(* CoDeSys 2.3 export: 6SHU-PV1.EXP *)

(* POU MAIN, CFC *)
PROGRAM MAIN
VAR
	TCT: ISTOK_TaskCycleTime;
END_VAR
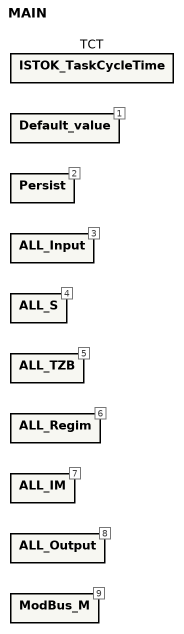
_CFC_ (* Continuous Function Chart, elements in execution order *)
#0 TCT:ISTOK_TaskCycleTime()
#1 Default_value()
#2 Persist()
#3 ALL_Input()
#4 ALL_S()
#5 ALL_TZB()
#6 ALL_Regim()
#7 ALL_IM()
#8 ALL_Output()
#9 ModBus_M()
_END_CFC_
(* the same logic as Structured Text *)
TCT();
Default_value();
Persist();
ALL_Input();
ALL_S();
ALL_TZB();
ALL_Regim();
ALL_IM();
ALL_Output();
ModBus_M();
END_PROGRAM

(* POU Lib/ISTOK_TaskCycleTime, CFC *)
FUNCTION_BLOCK ISTOK_TaskCycleTime
VAR_INPUT
END_VAR
VAR_OUTPUT
END_VAR
VAR
END_VAR
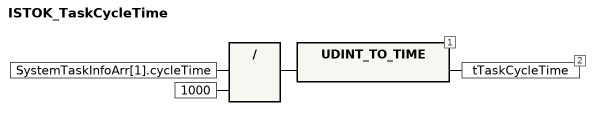
_CFC_ (* Continuous Function Chart, elements in execution order *)
#0 /(SystemTaskInfoArr[1].cycleTime, 1000)
#1 UDINT_TO_TIME(#0)
#2 tTaskCycleTime <= #1
_END_CFC_
END_FUNCTION_BLOCK

(* POU Default_value, CFC *)
PROGRAM Default_value
VAR
END_VAR
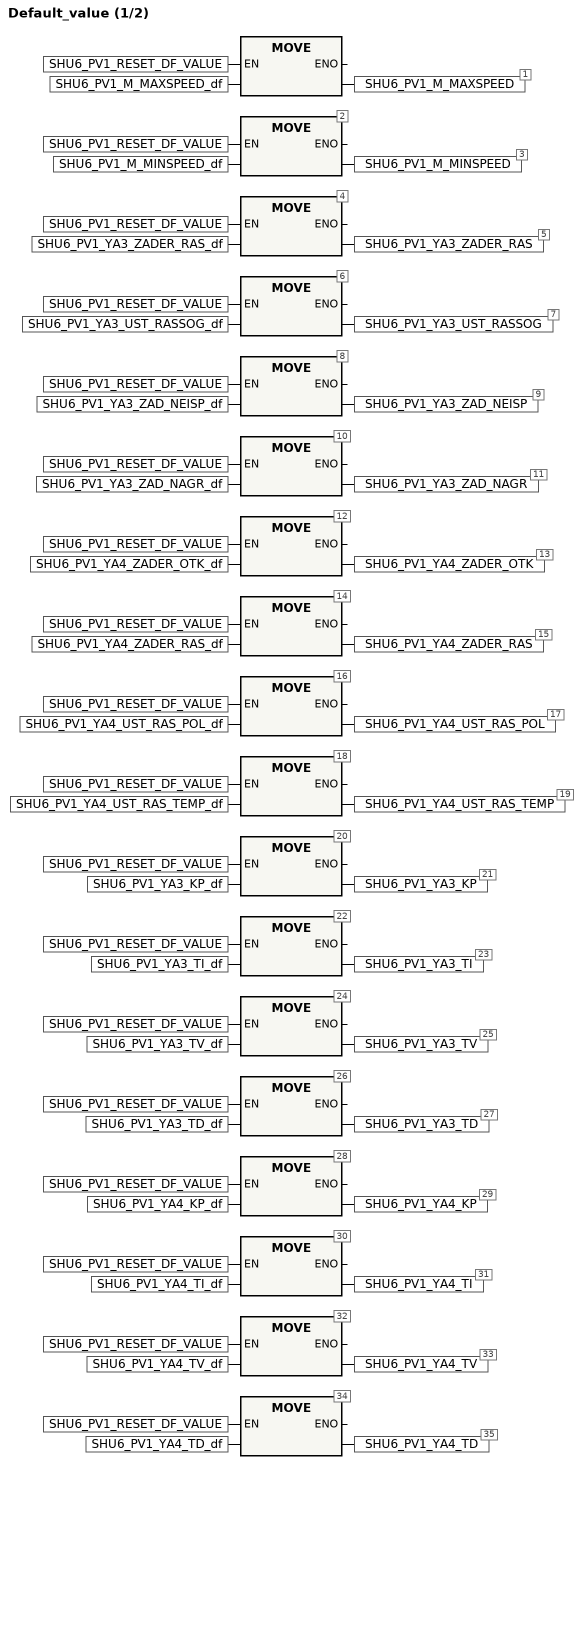
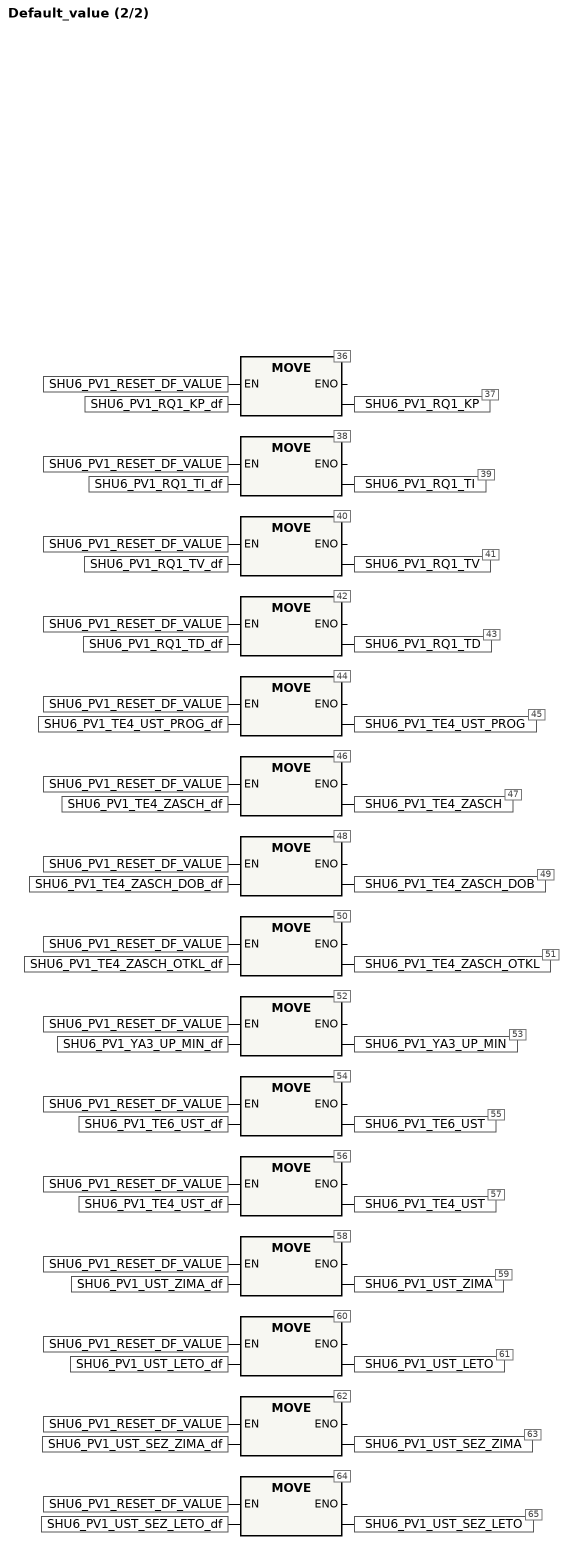
_CFC_ (* Continuous Function Chart, elements in execution order *)
#0 MOVE(EN: SHU6_PV1_RESET_DF_VALUE, SHU6_PV1_M_MAXSPEED_df)
#1 SHU6_PV1_M_MAXSPEED <= #0
#2 MOVE(EN: SHU6_PV1_RESET_DF_VALUE, SHU6_PV1_M_MINSPEED_df)
#3 SHU6_PV1_M_MINSPEED <= #2
#4 MOVE(EN: SHU6_PV1_RESET_DF_VALUE, SHU6_PV1_YA3_ZADER_RAS_df)
#5 SHU6_PV1_YA3_ZADER_RAS <= #4
#6 MOVE(EN: SHU6_PV1_RESET_DF_VALUE, SHU6_PV1_YA3_UST_RASSOG_df)
#7 SHU6_PV1_YA3_UST_RASSOG <= #6
#8 MOVE(EN: SHU6_PV1_RESET_DF_VALUE, SHU6_PV1_YA3_ZAD_NEISP_df)
#9 SHU6_PV1_YA3_ZAD_NEISP <= #8
#10 MOVE(EN: SHU6_PV1_RESET_DF_VALUE, SHU6_PV1_YA3_ZAD_NAGR_df)
#11 SHU6_PV1_YA3_ZAD_NAGR <= #10
#12 MOVE(EN: SHU6_PV1_RESET_DF_VALUE, SHU6_PV1_YA4_ZADER_OTK_df)
#13 SHU6_PV1_YA4_ZADER_OTK <= #12
#14 MOVE(EN: SHU6_PV1_RESET_DF_VALUE, SHU6_PV1_YA4_ZADER_RAS_df)
#15 SHU6_PV1_YA4_ZADER_RAS <= #14
#16 MOVE(EN: SHU6_PV1_RESET_DF_VALUE, SHU6_PV1_YA4_UST_RAS_POL_df)
#17 SHU6_PV1_YA4_UST_RAS_POL <= #16
#18 MOVE(EN: SHU6_PV1_RESET_DF_VALUE, SHU6_PV1_YA4_UST_RAS_TEMP_df)
#19 SHU6_PV1_YA4_UST_RAS_TEMP <= #18
#20 MOVE(EN: SHU6_PV1_RESET_DF_VALUE, SHU6_PV1_YA3_KP_df)
#21 SHU6_PV1_YA3_KP <= #20
#22 MOVE(EN: SHU6_PV1_RESET_DF_VALUE, SHU6_PV1_YA3_TI_df)
#23 SHU6_PV1_YA3_TI <= #22
#24 MOVE(EN: SHU6_PV1_RESET_DF_VALUE, SHU6_PV1_YA3_TV_df)
#25 SHU6_PV1_YA3_TV <= #24
#26 MOVE(EN: SHU6_PV1_RESET_DF_VALUE, SHU6_PV1_YA3_TD_df)
#27 SHU6_PV1_YA3_TD <= #26
#28 MOVE(EN: SHU6_PV1_RESET_DF_VALUE, SHU6_PV1_YA4_KP_df)
#29 SHU6_PV1_YA4_KP <= #28
#30 MOVE(EN: SHU6_PV1_RESET_DF_VALUE, SHU6_PV1_YA4_TI_df)
#31 SHU6_PV1_YA4_TI <= #30
#32 MOVE(EN: SHU6_PV1_RESET_DF_VALUE, SHU6_PV1_YA4_TV_df)
#33 SHU6_PV1_YA4_TV <= #32
#34 MOVE(EN: SHU6_PV1_RESET_DF_VALUE, SHU6_PV1_YA4_TD_df)
#35 SHU6_PV1_YA4_TD <= #34
#36 MOVE(EN: SHU6_PV1_RESET_DF_VALUE, SHU6_PV1_RQ1_KP_df)
#37 SHU6_PV1_RQ1_KP <= #36
#38 MOVE(EN: SHU6_PV1_RESET_DF_VALUE, SHU6_PV1_RQ1_TI_df)
#39 SHU6_PV1_RQ1_TI <= #38
#40 MOVE(EN: SHU6_PV1_RESET_DF_VALUE, SHU6_PV1_RQ1_TV_df)
#41 SHU6_PV1_RQ1_TV <= #40
#42 MOVE(EN: SHU6_PV1_RESET_DF_VALUE, SHU6_PV1_RQ1_TD_df)
#43 SHU6_PV1_RQ1_TD <= #42
#44 MOVE(EN: SHU6_PV1_RESET_DF_VALUE, SHU6_PV1_TE4_UST_PROG_df)
#45 SHU6_PV1_TE4_UST_PROG <= #44
#46 MOVE(EN: SHU6_PV1_RESET_DF_VALUE, SHU6_PV1_TE4_ZASCH_df)
#47 SHU6_PV1_TE4_ZASCH <= #46
#48 MOVE(EN: SHU6_PV1_RESET_DF_VALUE, SHU6_PV1_TE4_ZASCH_DOB_df)
#49 SHU6_PV1_TE4_ZASCH_DOB <= #48
#50 MOVE(EN: SHU6_PV1_RESET_DF_VALUE, SHU6_PV1_TE4_ZASCH_OTKL_df)
#51 SHU6_PV1_TE4_ZASCH_OTKL <= #50
#52 MOVE(EN: SHU6_PV1_RESET_DF_VALUE, SHU6_PV1_YA3_UP_MIN_df)
#53 SHU6_PV1_YA3_UP_MIN <= #52
#54 MOVE(EN: SHU6_PV1_RESET_DF_VALUE, SHU6_PV1_TE6_UST_df)
#55 SHU6_PV1_TE6_UST <= #54
#56 MOVE(EN: SHU6_PV1_RESET_DF_VALUE, SHU6_PV1_TE4_UST_df)
#57 SHU6_PV1_TE4_UST <= #56
#58 MOVE(EN: SHU6_PV1_RESET_DF_VALUE, SHU6_PV1_UST_ZIMA_df)
#59 SHU6_PV1_UST_ZIMA <= #58
#60 MOVE(EN: SHU6_PV1_RESET_DF_VALUE, SHU6_PV1_UST_LETO_df)
#61 SHU6_PV1_UST_LETO <= #60
#62 MOVE(EN: SHU6_PV1_RESET_DF_VALUE, SHU6_PV1_UST_SEZ_ZIMA_df)
#63 SHU6_PV1_UST_SEZ_ZIMA <= #62
#64 MOVE(EN: SHU6_PV1_RESET_DF_VALUE, SHU6_PV1_UST_SEZ_LETO_df)
#65 SHU6_PV1_UST_SEZ_LETO <= #64
_END_CFC_
(* the same logic as Structured Text *)
IF SHU6_PV1_RESET_DF_VALUE THEN SHU6_PV1_M_MAXSPEED := SHU6_PV1_M_MAXSPEED_df; END_IF;
IF SHU6_PV1_RESET_DF_VALUE THEN SHU6_PV1_M_MINSPEED := SHU6_PV1_M_MINSPEED_df; END_IF;
IF SHU6_PV1_RESET_DF_VALUE THEN SHU6_PV1_YA3_ZADER_RAS := SHU6_PV1_YA3_ZADER_RAS_df; END_IF;
IF SHU6_PV1_RESET_DF_VALUE THEN SHU6_PV1_YA3_UST_RASSOG := SHU6_PV1_YA3_UST_RASSOG_df; END_IF;
IF SHU6_PV1_RESET_DF_VALUE THEN SHU6_PV1_YA3_ZAD_NEISP := SHU6_PV1_YA3_ZAD_NEISP_df; END_IF;
IF SHU6_PV1_RESET_DF_VALUE THEN SHU6_PV1_YA3_ZAD_NAGR := SHU6_PV1_YA3_ZAD_NAGR_df; END_IF;
IF SHU6_PV1_RESET_DF_VALUE THEN SHU6_PV1_YA4_ZADER_OTK := SHU6_PV1_YA4_ZADER_OTK_df; END_IF;
IF SHU6_PV1_RESET_DF_VALUE THEN SHU6_PV1_YA4_ZADER_RAS := SHU6_PV1_YA4_ZADER_RAS_df; END_IF;
IF SHU6_PV1_RESET_DF_VALUE THEN SHU6_PV1_YA4_UST_RAS_POL := SHU6_PV1_YA4_UST_RAS_POL_df; END_IF;
IF SHU6_PV1_RESET_DF_VALUE THEN SHU6_PV1_YA4_UST_RAS_TEMP := SHU6_PV1_YA4_UST_RAS_TEMP_df; END_IF;
IF SHU6_PV1_RESET_DF_VALUE THEN SHU6_PV1_YA3_KP := SHU6_PV1_YA3_KP_df; END_IF;
IF SHU6_PV1_RESET_DF_VALUE THEN SHU6_PV1_YA3_TI := SHU6_PV1_YA3_TI_df; END_IF;
IF SHU6_PV1_RESET_DF_VALUE THEN SHU6_PV1_YA3_TV := SHU6_PV1_YA3_TV_df; END_IF;
IF SHU6_PV1_RESET_DF_VALUE THEN SHU6_PV1_YA3_TD := SHU6_PV1_YA3_TD_df; END_IF;
IF SHU6_PV1_RESET_DF_VALUE THEN SHU6_PV1_YA4_KP := SHU6_PV1_YA4_KP_df; END_IF;
IF SHU6_PV1_RESET_DF_VALUE THEN SHU6_PV1_YA4_TI := SHU6_PV1_YA4_TI_df; END_IF;
IF SHU6_PV1_RESET_DF_VALUE THEN SHU6_PV1_YA4_TV := SHU6_PV1_YA4_TV_df; END_IF;
IF SHU6_PV1_RESET_DF_VALUE THEN SHU6_PV1_YA4_TD := SHU6_PV1_YA4_TD_df; END_IF;
IF SHU6_PV1_RESET_DF_VALUE THEN SHU6_PV1_RQ1_KP := SHU6_PV1_RQ1_KP_df; END_IF;
IF SHU6_PV1_RESET_DF_VALUE THEN SHU6_PV1_RQ1_TI := SHU6_PV1_RQ1_TI_df; END_IF;
IF SHU6_PV1_RESET_DF_VALUE THEN SHU6_PV1_RQ1_TV := SHU6_PV1_RQ1_TV_df; END_IF;
IF SHU6_PV1_RESET_DF_VALUE THEN SHU6_PV1_RQ1_TD := SHU6_PV1_RQ1_TD_df; END_IF;
IF SHU6_PV1_RESET_DF_VALUE THEN SHU6_PV1_TE4_UST_PROG := SHU6_PV1_TE4_UST_PROG_df; END_IF;
IF SHU6_PV1_RESET_DF_VALUE THEN SHU6_PV1_TE4_ZASCH := SHU6_PV1_TE4_ZASCH_df; END_IF;
IF SHU6_PV1_RESET_DF_VALUE THEN SHU6_PV1_TE4_ZASCH_DOB := SHU6_PV1_TE4_ZASCH_DOB_df; END_IF;
IF SHU6_PV1_RESET_DF_VALUE THEN SHU6_PV1_TE4_ZASCH_OTKL := SHU6_PV1_TE4_ZASCH_OTKL_df; END_IF;
IF SHU6_PV1_RESET_DF_VALUE THEN SHU6_PV1_YA3_UP_MIN := SHU6_PV1_YA3_UP_MIN_df; END_IF;
IF SHU6_PV1_RESET_DF_VALUE THEN SHU6_PV1_TE6_UST := SHU6_PV1_TE6_UST_df; END_IF;
IF SHU6_PV1_RESET_DF_VALUE THEN SHU6_PV1_TE4_UST := SHU6_PV1_TE4_UST_df; END_IF;
IF SHU6_PV1_RESET_DF_VALUE THEN SHU6_PV1_UST_ZIMA := SHU6_PV1_UST_ZIMA_df; END_IF;
IF SHU6_PV1_RESET_DF_VALUE THEN SHU6_PV1_UST_LETO := SHU6_PV1_UST_LETO_df; END_IF;
IF SHU6_PV1_RESET_DF_VALUE THEN SHU6_PV1_UST_SEZ_ZIMA := SHU6_PV1_UST_SEZ_ZIMA_df; END_IF;
IF SHU6_PV1_RESET_DF_VALUE THEN SHU6_PV1_UST_SEZ_LETO := SHU6_PV1_UST_SEZ_LETO_df; END_IF;
END_PROGRAM

(* POU Persist, ST *)
PROGRAM Persist
VAR
	Save: WritePersistentData;
END_VAR
Save(NETID:='10.150.0.24.1.1',PORT:=801,START:=TRUE,TMOUT:=t#1s ,BUSY=> ,ERR=> ,	ERRID=> );
Save(NETID:='10.150.0.24.1.1',PORT:=801,START:= FALSE ,TMOUT:=t#1s ,BUSY=> ,ERR=> ,ERRID=> );
END_PROGRAM

(* POU Input/ALL_Input, CFC *)
PROGRAM ALL_Input
VAR
END_VAR
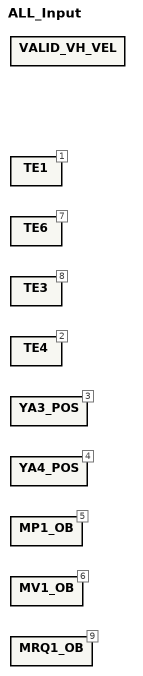
_CFC_ (* Continuous Function Chart, elements in execution order *)
#0 VALID_VH_VEL()
#1 TE1()
#2 TE4()
#3 YA3_POS()
#4 YA4_POS()
#5 MP1_OB()
#6 MV1_OB()
#7 TE6()
#8 TE3()
#9 MRQ1_OB()
_END_CFC_
(* the same logic as Structured Text *)
VALID_VH_VEL();
TE1();
TE4();
YA3_POS();
YA4_POS();
MP1_OB();
MV1_OB();
TE6();
TE3();
MRQ1_OB();
END_PROGRAM

(* POU Input/VALID_VH_VEL, CFC *)
PROGRAM VALID_VH_VEL
VAR
	RT_VKL_OLD_SEZ_LETO: R_TRIG;
         RT_VKL_OLD_SEZ_ZIMA: R_TRIG;

         SHU6_PV1_UST_SEZ_LETO_OLD: REAL;
	SHU6_PV1_UST_SEZ_ZIMA_OLD: REAL;

         SHU6_PV1_TE6_UST_OTKL_OLD: REAL;
	SHU6_PV1_TE6_UST_VKL_OLD: REAL;

         RT_TE6_UST_OTKL_OLD: R_TRIG;
         RT_TE6_UST_VKL_OLD: R_TRIG;
END_VAR
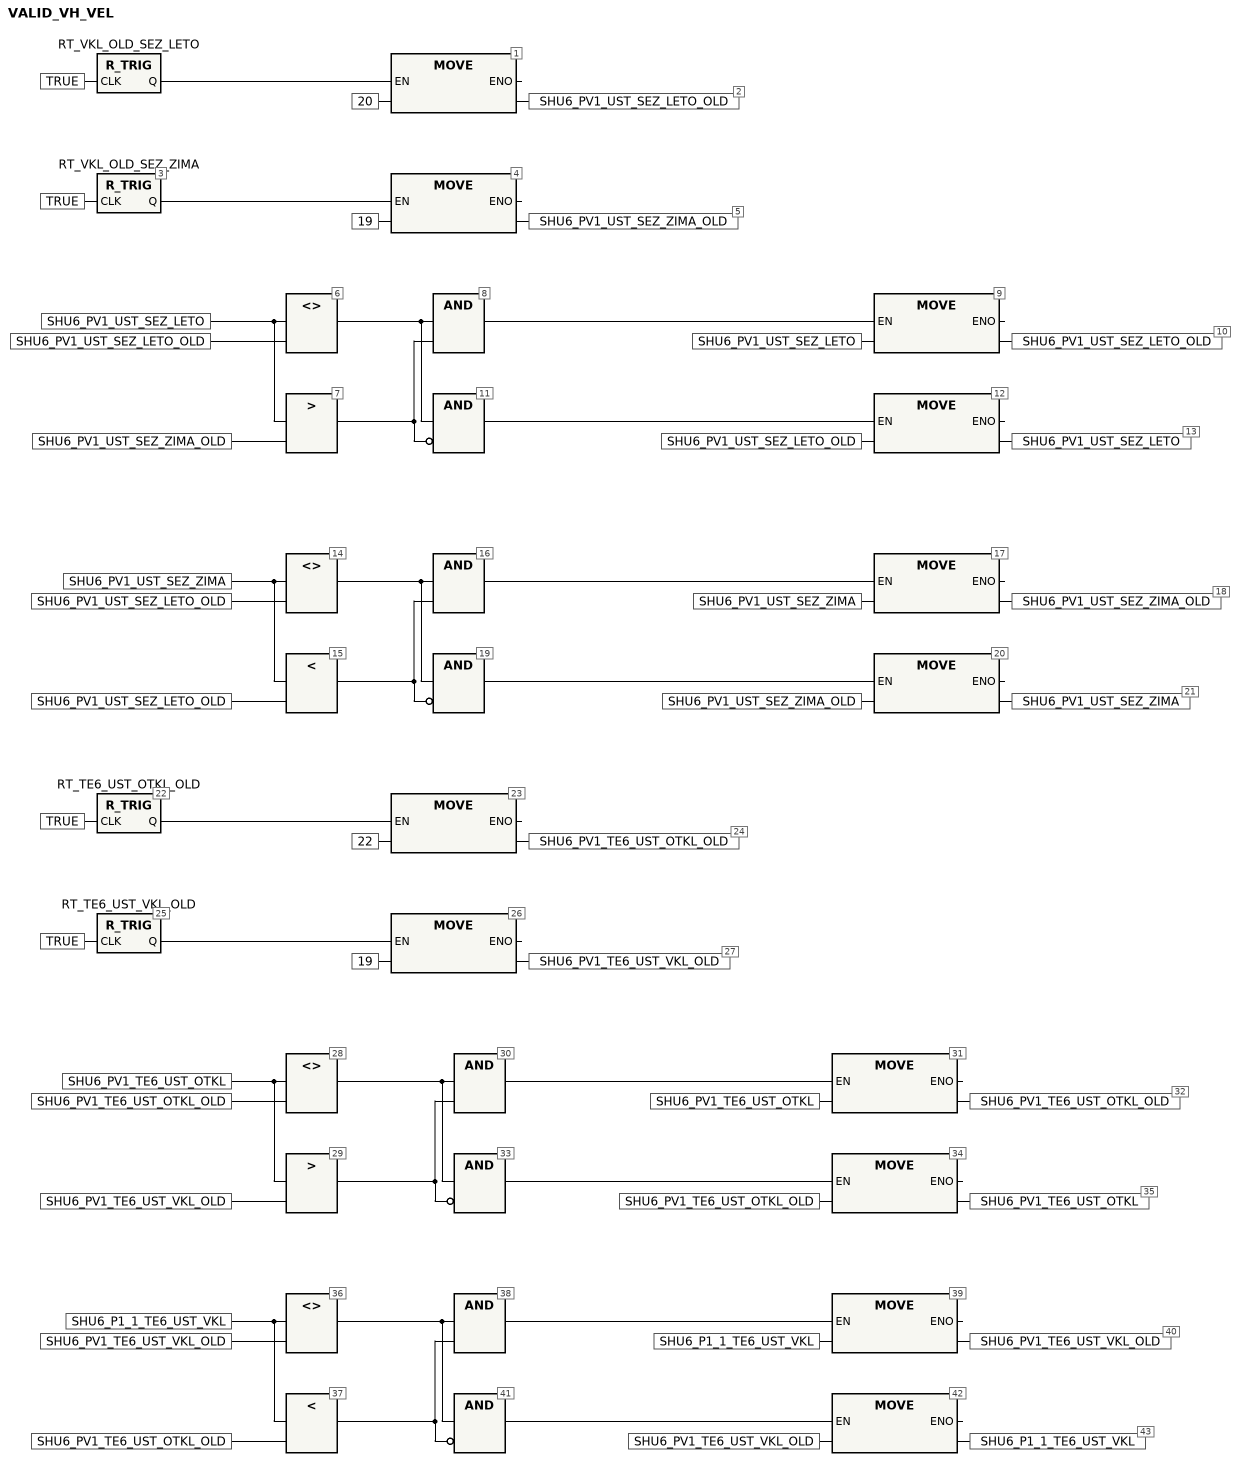
